FUNCTION_BLOCK Hysteresis
VAR_INPUT
	Val: REAL;
	OnVal: REAL;
	OffVal: REAL;
END_VAR
VAR_OUTPUT
	Out: BOOL;
END_VAR
VAR
END_VAR

IF Val < OffVal THEN
	Out := 0;
ELSIF Val > OnVal THEN
	Out := 1;
END_IF

END_FUNCTION_BLOCK

(* stored: Version 1.1.0.1, ProductVersion 3.1.4024.0
   POU Hysteresis: Id {e7dbce2b-3037-48fa-810a-c4124cd6b3cc}, SpecialFunc None *)
